(* IEC 61131-3 sources: Lasal/CPU_5344_V01/Class/RamSregels, 1 file *)

(* ---- RamSregels.st ---- *)
(*!
<Class
	Name               = "RamSregels"
	Revision           = "0.0"
	RealtimeTask       = "false"
	CyclicTask         = "false"
	BackgroundTask     = "false"
	Sigmatek           = "false"
	OSInterface        = "false"
	HighPriority       = "false"
	Automatic          = "false"
	UpdateMode         = "Prescan"
	SharedCommandTable = "true"
	Objectsize         = "(284,120)">
	<Channels>
		<Server Name="ClassSvr" Visualized="false" Initialize="false" WriteProtected="true" Retentive="false"/>
	</Channels>
</Class>
*)
RamSregels : CLASS
  //Servers:
	ClassSvr 	: SvrChCmd_DINT;
  //Clients:
  //Variables:
		Sregels 	: SRegelInfoArray;
  //Functions:

	FUNCTION GLOBAL givePtr
		VAR_OUTPUT
			Ptr 	: ^USINT;
		END_VAR;

	FUNCTION GLOBAL ReadLine
		VAR_INPUT
			Nr 	: DINT;
		END_VAR
		VAR_OUTPUT
			Regel 	: SRegelInfo;
		END_VAR;

	FUNCTION GLOBAL WriteLine
		VAR_INPUT
			Nr 	: DINT;
			Regel 	: SRegelInfo;
		END_VAR;

	FUNCTION GLOBAL ClearAll;

	FUNCTION GLOBAL ReadTable
		VAR_OUTPUT
			tabel 	: SRegelInfoArray;
		END_VAR;

	FUNCTION GLOBAL WriteTable
		VAR_INPUT
			tabel 	: SRegelInfoArray;
		END_VAR;
  //Tables:
	FUNCTION @STD
		VAR_OUTPUT
			ret_code	: CONFSTATES;
		END_VAR;
	FUNCTION GLOBAL TAB @CT_;
END_CLASS;

FUNCTION GLOBAL RamSregels::givePtr
	VAR_OUTPUT
		Ptr 	: ^USINT;
	END_VAR

  Ptr := #Sregels$USINT;

END_FUNCTION

FUNCTION GLOBAL RamSregels::ReadLine
	VAR_INPUT
		Nr 	: DINT;
	END_VAR
	VAR_OUTPUT
		Regel 	: SRegelInfo;
	END_VAR

  Regel := Sregels[Nr];

END_FUNCTION

FUNCTION GLOBAL RamSregels::WriteLine
	VAR_INPUT
		Nr 	: DINT;
		Regel 	: SRegelInfo;
	END_VAR
  //max nr is in class hiervoor geregeld
  Sregels[Nr] := Regel;

END_FUNCTION

FUNCTION GLOBAL RamSregels::ClearAll

  _memset(dest:=#Sregels[0], usByte:=0, cntr:=sizeof(Sregels));

END_FUNCTION

FUNCTION GLOBAL RamSregels::ReadTable
	VAR_OUTPUT
		tabel 	: SRegelInfoArray;
	END_VAR

  tabel := Sregels;

END_FUNCTION

FUNCTION GLOBAL RamSregels::WriteTable
	VAR_INPUT
		tabel 	: SRegelInfoArray;
	END_VAR

  Sregels := tabel;

END_FUNCTION
